PROGRAM MedidaTempTarjeta
VAR
END_VAR

GVL.TempTerB:=IO.I_TermB/10.0;

GVL.TempTerT:=IO.I_TermT/10.0;

END_PROGRAM

(* stored: Version 1.1.0.1, ProductVersion 3.1.4024.9
   POU MedidaTempTarjeta: Id {f19342b6-768b-4a38-8450-104223824197}, SpecialFunc None *)
